VAR_GLOBAL
	RemoverPartPresent	:	BOOL;
	Remover	:	BOOL;
END_VAR

(* stored: Version 1.1.0.1
   GVL Remover: Id {7d463467-d51e-4781-88b6-5ca11176fe60} *)
